{attribute 'qualified_only'}
{attribute 'strict'}
TYPE E_MOTOR_MOVE_TYPE :
(
	NONE	:= 0,
	
	ABSOLUTE,
	RELATIVE,
	VELOCITY,
	TRACKING

);
END_TYPE

(* stored: Version 1.1.0.1, ProductVersion 3.1.4022.16
   DUT E_MOTOR_MOVE_TYPE: Id {83f74184-8f65-4c01-a3ab-b6eb019f7a1e} *)
